KUKA KRL program: MacroReadMe.src

&ACCESS RVP
&COMMENT ReadMe File
DEF  MacroReadMe ( )

; This file only exists as a directory placeholder file.

END
